{attribute 'linkalways'} 
{attribute 'no_explicit_call' := 'This FB is a CLASS and must be accessed using methods or properties'}
{attribute 'enable_dynamic_creation'}
FUNCTION_BLOCK Node_F_VN_RotatedRectangleCorners EXTENDS VisionNode
VAR
    stRect : _TcVnRotatedRectangle;
    aCorners : _TcVnArray4_Point2_REAL;
    hrPrev : _HRESULT(S_OK);
	hresult : _HRESULT(S_OK);
END_VAR

METHOD PUBLIC  Clone : I_Node
VAR
	pNode : POINTER TO Node_F_VN_RotatedRectangleCorners;
END_VAR
pNode := __NEW(Node_F_VN_RotatedRectangleCorners);
Clone := pNode^;
END_METHOD

METHOD FB_init : BOOL
VAR_INPUT
	bInitRetains : BOOL; // if TRUE, the retain variables are initialized (warm start / cold start)
	bInCopyCode : BOOL;  // if TRUE, the instance afterwards gets moved into the copy code (online change)
END_VAR
AddInput('stRect', stRect);
AddInput('hrPrev', hrPrev);
AddOutput('aCorners', aCorners);
AddOutput('hresult',hresult);
END_METHOD

METHOD PROTECTED OnExecute
hresult.Value := F_VN_RotatedRectangleCorners(
    stRect := stRect.Value,
    aCorners := aCorners.Value,
	hrPrev:= hrPrev.Value);
END_METHOD

METHOD PUBLIC PreExecutionCheck
VAR_INPUT
	Check : I_PreExecutionChecks;
END_VAR
END_METHOD

END_FUNCTION_BLOCK

(* stored: Version 1.1.0.1, ProductVersion 3.1.4024.13
   POU Node_F_VN_RotatedRectangleCorners: Id {7e3a62be-8443-00a4-36ed-3bc881f26a36}, SpecialFunc None
   Folder Constructor: Id {fbd8d76a-49d8-0820-1d99-6593a6b51d89}
   Method Clone: Id {e61c3806-651a-0f74-1226-72d48201a346}
   Method FB_init: Id {cc1b7184-557c-00ec-2956-a65fecbd3df1}
   Method OnExecute: Id {ddb380d9-784c-0807-1376-91e705845025}
   Method PreExecutionCheck: Id {7d1bb589-4765-0f23-29ab-2b618f1921de} *)
